TYPE ST_VarSetCmd :
STRUCT
	ArrayType: DUT_Command_ArrayType;
	ArrayIndex: INT;
	Coordinates: DUT_COORD_REF;
END_STRUCT
END_TYPE

(* stored: Version 1.1.0.1
   DUT ST_VarSetCmd: Id {0b1a37a4-4123-4a33-84fb-db1ab5afd1a7} *)
